TEXTLIST TL_Frames
  0 = 'Home' | EN\: 'Home' | PL: 'Główna'
  1 = 'Alarms' | EN\: 'Alarms' | PL: 'Alarmy'
  2 = 'Info' | EN\: 'Info' | PL: 'Info'
  3 = 'Users' | EN\: 'Users' | PL: 'Użytkownicy'
  4 = 'Settings' | EN\: 'Settings' | PL: 'Ustawienia'
  5 = 'File Dialog' | EN\: 'File Dialog' | PL: 'Dialog plików'
  6 = 'Table' | EN\: 'Table' | PL: 'Tabela'
  7 = 'Trends' | EN\: 'Trends' | PL: 'Trendy'
  8 = 'Option4' | EN\: 'Option4' | PL: 'Opcja4'
  9 = 'Option5' | EN\: 'Option5' | PL: 'Opcja5'
  10 = 'Option6' | EN\: 'Opion6' | PL: 'Opcja6'
   = ''
END_TEXTLIST

(* stored: Version 1.1.0.1, ProductVersion 3.1.4022.6
   TextList TL_Frames: Id {63b0673b-cd4d-4bfd-893f-bb607e749546} *)
